FUNCTION_BLOCK UA_MethodCall_ADSReadReq
VAR_INPUT
	bExecute			: BOOL;
	nConnectionHdl		: DWORD;
	nNamespaceIndex		: UINT; 			(* to be retrieved using UA_GetNamespaceIndex *)
	sNetID				: T_AmsNetId; 		(* AmsNetId OF the Target *)
	nPort				: INT; 				(* Port number	*)
	nIndexGroup			: DINT;				(* IndexGroup*)
	nIndexOffset		: DINT; 			(* IndexOffset*)
	pOutputArgInfoAndData	: PVOID;
	cbOutputArgInfoAndData	: UDINT;			(* Count of bytes to be read*)
	cbReadData			: UDINT;			(* Count of bytes to be read*)
	nNumberOfOutputArguments	: UDINT; 
	pOutputArgInfo		: POINTER TO ST_UAMethodArgInfo; 
	cbOutputArgInfo		: UDINT;
	Timeout				: TIME := DEFAULT_ADS_TIMEOUT;
END_VAR
VAR_OUTPUT
	cbReadData_R		: UDINT;			(* Count of bytes to be read*)
	bDone				: BOOL;
	bBusy				: BOOL;
	bError				: BOOL;
	nErrorID			: DWORD;
END_VAR
VAR
	iReadReqState			: INT;
	RTrig					: R_TRIG;

	fbUA_MethodGetHandle	: UA_MethodGetHandle;
	nMethodHdl				: DWORD;
	ObjectNodeID			: ST_UANodeID;
	MethodNodeID			: ST_UANodeID;

	fbUA_MethodCall			: UA_MethodCall;
	InputArguments			: ARRAY [1..nNumberOfInputArguments] OF ST_UAMethodArgInfo; (*ReadReq has 5 input parameters *)
	
	nArg					: INT;
	fbUA_MethodReleaseHandle: UA_MethodReleaseHandle;

	nInputData			: ARRAY [1..nInputArgSize] OF BYTE; (* NetID(24)+ Port(2)+ IG(4)+ IO(4)+ cbData(4)*)
	nOffset				: UDINT;
	bInputDataError		: BOOL;
END_VAR
VAR CONSTANT
	nInputArgSize			: UDINT := 38; (* NetID(24)+ Port(2)+ IG(4)+ IO(4)+ cbData(4)*)
	nNumberOfInputArguments : UDINT := 5;
END_VAR

(*
ADSReadReq(
******** Input Arguments ********
	string24 sNetID, 		: AmsNetId of the Target
	int16 Port,			: Port number	
	int32 IndexGroup,		: IndexGroup
	int32 IndexOffset,		: IndexOffset
	uint32 cbData			: Count of bytes to be read
******** Output Arguments ********
	bytestring Data		: Data read from device
);

*)
RTrig(CLK:= bExecute);

CASE iReadReqState OF

0:	(* Get Method Handle *)
	IF RTrig.Q THEN
		bBusy	:= TRUE;
		bDone 	:= FALSE;
		bError	:= FALSE;
		nErrorID	:= 0;
		ObjectNodeID.eIdentifierType 	:= eUAIdentifierType_String;
		ObjectNodeID.nNamespaceIndex 	:= nNamespaceIndex;
		ObjectNodeID.sIdentifier		:= 'ADSAMS';
	
		MethodNodeID.eIdentifierType 	:= eUAIdentifierType_String;
		MethodNodeID.nNamespaceIndex 	:= nNamespaceIndex;
		MethodNodeID.sIdentifier		:= 'ADSAMS.AdsReadReq';

		M_Init();
		IF bInputDataError = FALSE THEN
			iReadReqState 	:= iReadReqState + 1;
		ELSE
			bBusy 		:= FALSE; 
			bError 		:= TRUE;
			nErrorID 	:= DEVICE_INVALIDSIZE; //16#705 parameter size not correct
		END_IF
		
	END_IF


1:	(* Method Get Handle *)
	fbUA_MethodGetHandle(
			Execute			:= TRUE,
			ConnectionHdl	:= nConnectionHdl,
			ObjectNodeID	:= ObjectNodeID,
			MethodNodeID 	:= MethodNodeID,
			Timeout			:= Timeout,
			MethodHdl		=> nMethodHdl
		);
	IF NOT fbUA_MethodGetHandle.Busy THEN
		fbUA_MethodGetHandle(Execute := FALSE);

		IF NOT fbUA_MethodGetHandle.Error THEN
			(*  *)
			iReadReqState 	:= iReadReqState + 1; (* Call Method *)
		ELSE
			bError		:= TRUE;
			nErrorID		:= fbUA_MethodGetHandle.ErrorID;
			iReadReqState 	:= 3; (* Release Handle *)
		END_IF
	END_IF


2:	(* Method Call *)
	fbUA_MethodCall(
		Execute					:= TRUE,
		ConnectionHdl			:= nConnectionHdl,
		MethodHdl				:= nMethodHdl,
		nNumberOfInputArguments := nNumberOfInputArguments, (* 5 *)
		pInputArgInfo			:= ADR(InputArguments),
		cbInputArgInfo			:= SIZEOF(InputArguments),
		pInputArgData			:= ADR(nInputData),
		cbInputArgData			:= nOffset,
		pInputWriteData			:= 0,		
		cbInputWriteData		:= 0,
		nNumberOfOutputArguments:= nNumberOfOutputArguments, (* input parameter: to be assigned by customer *)
		pOutputArgInfo			:= pOutputArgInfo,
		cbOutputArgInfo			:= cbOutputArgInfo,
		pOutputArgInfoAndData	:= pOutputArgInfoAndData,
		cbOutputArgInfoAndData	:= cbOutputArgInfoAndData,
		Timeout					:= Timeout
	);

	IF NOT fbUA_MethodCall.Busy THEN
		fbUA_MethodCall(Execute := FALSE, cbRead_R => cbReadData_R);

		IF NOT fbUA_MethodCall.Error THEN
			(*  *)
			iReadReqState 	:= iReadReqState + 1; (* Release handle *)
		ELSE
			bError		:= TRUE;
			nErrorID		:= fbUA_MethodCall.ErrorID;
			iReadReqState 	:= 3; (* Release handle *)
		END_IF
	END_IF


3:	(* Release Method Handle *)
	fbUA_MethodReleaseHandle(
		Execute			:= TRUE,
		ConnectionHdl	:= nConnectionHdl,
		MethodHdl		:= nMethodHdl,
		Timeout			:= Timeout
	);

	IF NOT fbUA_MethodReleaseHandle.Busy THEN
		fbUA_MethodReleaseHandle(Execute := FALSE);
		bBusy := FALSE;
		IF NOT fbUA_MethodReleaseHandle.Error THEN
			(* session closed *)
			bDone := TRUE;
			iReadReqState 	:= 0; (* idle *)
		ELSE
			bError			:= TRUE;
			nErrorID		:= fbUA_MethodReleaseHandle.ErrorID;
			iReadReqState 	:= 0; (* idle *)
		END_IF
	END_IF
END_CASE

ACTION M_Init:
bInputDataError := FALSE; 
nOffset := 0;
MEMSET(ADR(InputArguments),0,SIZEOF(InputArguments));
MEMSET(ADR(nInputData),0,SIZEOF(nInputData));

nArg := 1;
(*sNetID := sAmsNetID;*)		(********** NET ID **********)
InputArguments[nArg].DataType			:= eUAType_String;
InputArguments[nArg].ValueRank			:= -1; 							(* Scalar or Array *)
InputArguments[nArg].ArrayDimensions[1]	:= 0; 							(* Number of Dimension in case its an array *)
InputArguments[nArg].nLenData			:= INT_TO_UDINT(LEN(sNetId)) + 1;				(* Length if its a STRING *)
IF nOffset + INT_TO_UDINT(LEN(sNetId))+1 > nInputArgSize THEN 
	bInputDataError := TRUE;
	RETURN;
ELSE
	MEMCPY(ADR(nInputData)+nOffset,ADR(sNetId),INT_TO_UDINT(LEN(sNetId))+1);				(* VALUE in BYTES FORM *)
	nOffset := nOffset + INT_TO_UDINT(LEN(sNetId))+1;
END_IF

nArg := nArg + 1;
(* nPort := 851;*)			(********** PORT **********)
InputArguments[nArg].DataType			:= eUAType_Int16;
InputArguments[nArg].ValueRank			:= -1; 							(* Scalar or Array *)
InputArguments[nArg].ArrayDimensions[1]	:= 0; 							(* Number of Dimension in case its an array *)
InputArguments[nArg].nLenData			:= SIZEOF(nPort);				(* Length if its a STRING *)
IF nOffset + SIZEOF(nPort) > nInputArgSize THEN 
	bInputDataError := TRUE;
	RETURN;
ELSE
	MEMCPY(ADR(nInputData)+nOffset,ADR(nPort),SIZEOF(nPort));			(* VALUE in BYTES FORM *)
	nOffset := nOffset + SIZEOF(nPort);
END_IF

nArg := nArg + 1;
(*nIndexGroup := 16#4020;*)	(********** INDEX GROUP **********)
InputArguments[nArg].DataType			:= eUAType_Int32;
InputArguments[nArg].ValueRank			:= -1; 							(* Scalar or Array *)
InputArguments[nArg].ArrayDimensions[1]	:= 0; 							(* Number of Dimension in case its an array *)
InputArguments[nArg].nLenData			:= SIZEOF(nIndexGroup);			(* Length if its a STRING *)
IF nOffset + SIZEOF(nIndexGroup) > nInputArgSize THEN 
	bInputDataError := TRUE;
	RETURN;
ELSE
	MEMCPY(ADR(nInputData)+nOffset,ADR(nIndexGroup),SIZEOF(nIndexGroup));		(* VALUE in BYTES FORM *)
	nOffset := nOffset + SIZEOF(nIndexGroup);
END_IF

nArg := nArg + 1;
(*nIndexOffset := 0; *)		(********** INDEX OFFSET **********)
InputArguments[nArg].DataType			:= eUAType_Int32;
InputArguments[nArg].ValueRank			:= -1; 							(* Scalar or Array *)
InputArguments[nArg].ArrayDimensions[1]	:= 0; 							(* Number of Dimension in case its an array *)
InputArguments[nArg].nLenData			:= SIZEOF(nIndexOffset);		(* Length if its a STRING *)
IF nOffset + SIZEOF(nIndexOffset) > nInputArgSize THEN 
	bInputDataError := TRUE;
	RETURN;
ELSE
	MEMCPY(ADR(nInputData)+nOffset,ADR(nIndexOffset),SIZEOF(nIndexOffset));	(* VALUE in BYTES FORM *)
	nOffset := nOffset + SIZEOF(nIndexOffset);
END_IF

nArg := nArg + 1;
(*nReadLength := 2; *)		(*********** ReadLength ***********)
InputArguments[nArg].DataType			:= eUAType_UInt32;
InputArguments[nArg].ValueRank			:= -1; 							(* Scalar or Array *)
InputArguments[nArg].ArrayDimensions[1]	:= 0; 							(* Number of Dimension in case its an array *)
InputArguments[nArg].nLenData			:= SIZEOF(cbReadData);	
IF nOffset + SIZEOF(cbReadData) > nInputArgSize THEN 
	bInputDataError := TRUE;
	RETURN;
ELSE			(* Length if its a STRING *)
	MEMCPY(ADR(nInputData)+nOffset,ADR(cbReadData),SIZEOF(cbReadData));				(* VALUE in BYTES FORM *)
	nOffset := nOffset + SIZEOF(cbReadData);
END_IF
END_ACTION

END_FUNCTION_BLOCK

(* stored: Version 1.1.0.1, ProductVersion 3.1.4022.6
   POU UA_MethodCall_ADSReadReq: Id {f57fd503-ac42-4557-8ee4-d8e4a42022c8}, SpecialFunc None
   Action M_Init: Id {ce3b7c65-bf68-4a6a-a949-8a9b17c5cdad} *)
